	FUNCTION_BLOCK FB 347
	TITLE =G247M LOCAL COMMAND BUTTON / LAMPS GERM 8
	//COPYRIGHT:    (C) 2009  BUHLER AG, CH-9240 UZWIL, SWITZERLAND
	//
	//PRODUCT:      WinCoS_BIW01_09
	//
	//TITLE:        LOCAL COMMAND BUTTON / LAMPS GERM 8
	//                Machine group control
	//                Maschinengruppensteuerung
	//
	//--------------------------------------------------------------------------------
	//
	//IDENT:        AUTHOR:             DEPT:                              DATE:
	//
	//P01_FB347.1.0 K.Renz              CSB41                              13.Jan.2010
	//             1st Release
	//
	//--------------------------------------------------------------------------------
	//
	//PURPOSE:
	//
	//MANUAL :
	//
	//RESTRICTIONS:
	//
	//--------------------------------------------------------------------------------
	AUTHOR  : KR
	FAMILY  : USW
	VERSION : 9.9


	VAR
	  Gr       : FB10;	//Standard interface to group
	  InOutValue1    : DINT; //Data for user
	  InOutValue2    : DINT; //Data for user
	  OutWayConflict : BOOL;	//Data for user
	  OutSelectionOk : BOOL;	//Data for user
	  CmdNewValue : BOOL;	//Data for user
	  CmdNewJob   : BOOL;	//Data for user
	  OutCodeOK   : BOOL;	//Data for user
	  InEndOfJob  : BOOL ;	//Data for user
	  staWayOk      : BOOL ;	//Data for user
	  EdgeStartRelease : BOOL ;	//Data for user
	  USW8  : BOOL;	//Data for user
	  USW9 : BOOL;	//Data for user
	  USW10: BOOL;	//Data for user
	  USW11: BOOL;	//Data for user
	  USW12: BOOL;	//Data for user
	  USW13: BOOL;	//Data for user
	  USW14: BOOL;	//Data for user
	  USW15: BOOL;	//Data for user
	     #A_2811_KCL01I1 : FB14;   // DigInpCont
	     #A_2811_KCL01I2 : FB14;   // DigInpCont
	     #A_2811_KCL01I3 : FB14;   // DigInpCont
	     #A_2811_KCL01I4 : FB14;   // DigInpCont
	     #A_2811_KCL01I5 : FB14;   // DigInpCont
	     #A_2811_KCL01I6 : FB14;   // DigInpCont
	     #A_2811_KCL01O1 : FB11;   // DigOut
	     #A_2811_KCL01O2 : FB11;   // DigOut
	     #A_2815_KCL01I1 : FB14;   // DigInpCont
	     #A_2815_KCL01I2 : FB14;   // DigInpCont
	     #A_2815_KCL01I3 : FB14;   // DigInpCont
	     #A_2815_KCL01I4 : FB14;   // DigInpCont
	     #A_2815_KCL01I5 : FB14;   // DigInpCont
	     #A_2815_KCL01I6 : FB14;   // DigInpCont
	     #A_2815_KCL01I7 : FB14;   // DigInpCont
	     #A_2815_KCL01I8 : FB14;   // DigInpCont
	     #A_2815_KCL01I9 : FB14;   // DigInpCont
	     #A_2815_KCL01O1 : FB11;   // DigOut
	     #A_2815_KCL01O2 : FB11;   // DigOut
	     #A_2815_KCL01O3 : FB11;   // DigOut
	     #A_2815_KCL01O4 : FB11;   // DigOut
	     #A_2815_KCL01O5 : FB11;   // DigOut
	     #A_2815_KCL01O6 : FB11;   // DigOut
	     #A_2815_KCL01O7 : FB11;   // DigOut
	END_VAR
	VAR_TEMP
	   tmpEnable		: BOOL;
	   tmpFlag  		: BOOL;
	   tmpCmdNext		: BOOL;
	   tmpLocal  		: BOOL;
	   tmpAspOk  		: BOOL;
	   tmpHWStop 		: BOOL;
	   tmpInstanzDBNo       : INT ;
	END_VAR
	BEGIN
	NETWORK
	TITLE =
	NETWORK
	TITLE =Read command from group control
	//Parameter
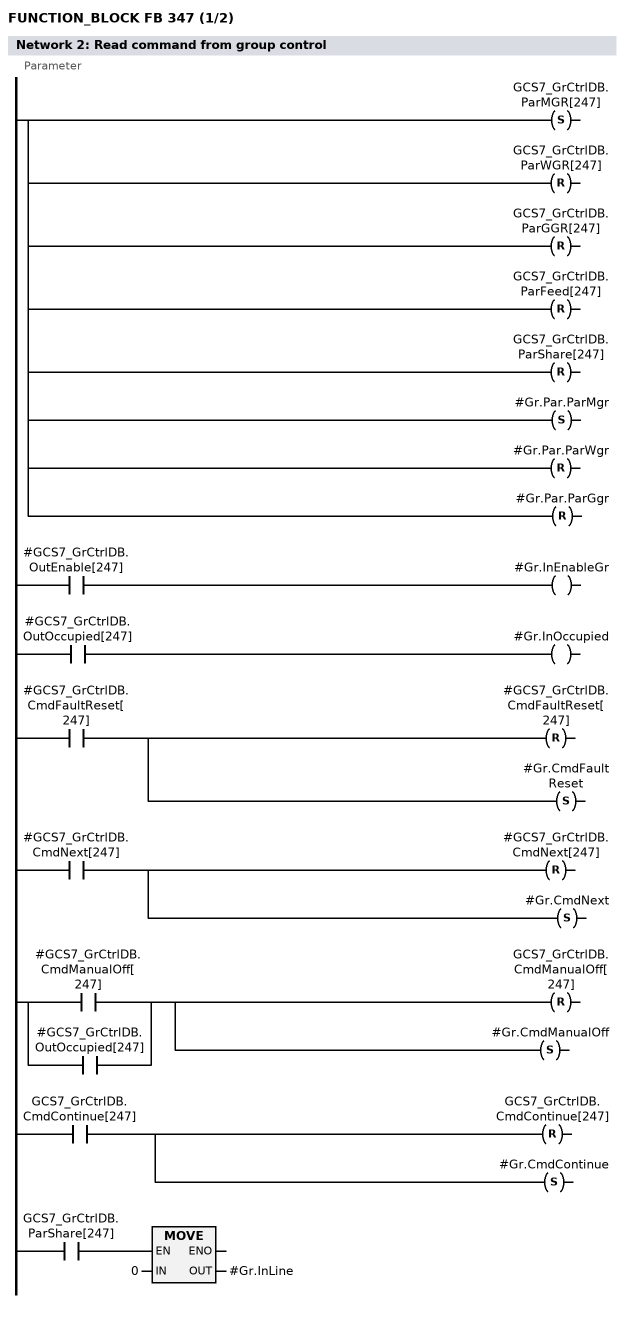
	      SET;
	      S   GCS7_GrCtrlDB.ParMGR[247];
	      R   GCS7_GrCtrlDB.ParWGR[247];
	      R   GCS7_GrCtrlDB.ParGGR[247];
	      R   GCS7_GrCtrlDB.ParFeed[247];
	      R   GCS7_GrCtrlDB.ParShare[247];
	      S   #Gr.Par.ParMgr;
	      R   #Gr.Par.ParWgr;
	      R   #Gr.Par.ParGgr;
	//Command
	      U   #GCS7_GrCtrlDB.OutEnable[247];
	      =   #Gr.InEnableGr;
	      U   #GCS7_GrCtrlDB.OutOccupied[247];
	      =   #Gr.InOccupied;
	      U   #GCS7_GrCtrlDB.CmdFaultReset[247];
	      R   #GCS7_GrCtrlDB.CmdFaultReset[247];
	      S   #Gr.CmdFaultReset;
	      U  #GCS7_GrCtrlDB.CmdNext[247];
	      R   #GCS7_GrCtrlDB.CmdNext[247];
	      S   #Gr.CmdNext;
	      U   #GCS7_GrCtrlDB.CmdManualOff[247];
	      O   #GCS7_GrCtrlDB.OutOccupied[247];
	      R   GCS7_GrCtrlDB.CmdManualOff[247];
	      S   #Gr.CmdManualOff;
	      U  GCS7_GrCtrlDB.CmdContinue[247];
	      R   GCS7_GrCtrlDB.CmdContinue[247];
	      S   #Gr.CmdContinue;
	//Init Line Number
	      U   GCS7_GrCtrlDB.ParShare[247];
	      SPBN WE00;
	      L     0;
	      T     #Gr.InLine;
	WE00: NOP   0;
	NETWORK
	TITLE =Call Methode Control
	// 1. Handle Interface PCControl
	// 2. Prepare mode --> ModePassive,ModeActive,ModeIdling
	// 3. Reset global flags of the group
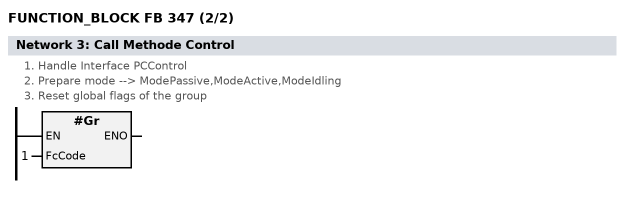
	      CALL #Gr (
	           FcCode                   := 1);
	NETWORK
	TITLE =Restart Idling Time
		L  #Gr.Par.ParIdling;
		L  2;
		>=I;
		SPB IdTm;
		T  #Gr.Par.ParIdling;
	IdTm:   NOP 0;
	      CLR;
	      S    #Gr.CmdRestartIdling;
	NETWORK
	TITLE =Prepare global flags
	NETWORK
	TITLE =Set Pattern (Target position)
	NETWORK
	TITLE =Interlocking WayOk
	//
	NETWORK
	TITLE =Interlocking Autostart
		CLR;
		R   #Gr.OutAutostart;
	NETWORK
	TITLE =Interlocking Enable
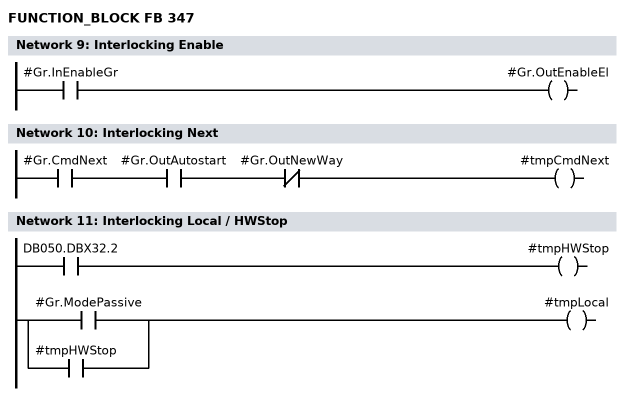
	      U     #Gr.InEnableGr;
	      =     #Gr.OutEnableEl;

	NETWORK
	TITLE =Interlocking Next
	      U     #Gr.CmdNext;
	      U     #Gr.OutAutostart;
	      UN    #Gr.OutNewWay;
	      =    #tmpCmdNext;

	NETWORK
	TITLE =Interlocking Local / HWStop
	      U    DB050.DBX32.2;
	      =    #tmpHWStop;

	      U    #Gr.ModePassive;
	      O    #tmpHWStop;
	      =    #tmpLocal;

	NETWORK
	TITLE =Interlocking Start Warning
	      NOP 0;
	//- Restart after fault --
	      U     #Gr.CmdFaultReset;
	      U     #Gr.VarFault;
	      S       "SYS_StartWarningDB".Area[9].CmdResetStartWarning;
	//- Run Timer --
	      AUF "G247M";
	      CALL  FB100 , DB100(
	       InModeHigher :=FALSE,
	       InArea     :=9,
	       InEnable   :=#Gr.OutEnableEl,
	       InLocal    :=#tmpLocal,
	       InStarted  :=#Gr.VarStarted,
	       InCmdNext  :=#tmpCmdNext,
	       OutCmdNext :=#tmpCmdNext,
	       OutStartwarning:=#Gr.VarStartWarning);
	//- Store Startwarning done  --
	//- Reset Autostart --
	      U     "SYS_StartWarningDB".TmpArea.OutStartReleaseRunningL;
	      FN    #EdgeStartRelease;
	      U     #Gr.VarFault;
	      R     #Gr.OutAutostart;
	NETWORK
	TITLE ==A-2811-KCL01I1 : SCREW ON BUTTON
	NOP 0;
	//-InLocal---
	      U     #tmpLocal;
	      =     #A_2811_KCL01I1.InLocal;
	//
	//-Monitoring---
	      CLR;
	      =      #A_2811_KCL01I1.InMonTrue;
	      CLR;
	      =      #A_2811_KCL01I1.InMonFalse;
	//
	//-PreAlarm---
	      CLR;
	      =      #A_2811_KCL01I1.InPreAlarmTrue;
	      CLR;
	      =      #A_2811_KCL01I1.InPreAlarmFalse;
	//
	//-Additional commands---
	//      CLR
	//      S     #A_2811_KCL01I1.CmdRunTimeOutTime
	//
	//-Read inputs---
	      U     E 840.4;
	      =     #A_2811_KCL01I1.InpTrue;
	      U   DB050.DBX32.2;
	      =     #A_2811_KCL01I1.InHWStop;
	       U     PLC_DPInfo.Master[1].SlavesError[84];
	       =       #A_2811_KCL01I1.InDPFault;
	//
	//-Set Parameters---
	//
	//-Call object control---
	      CALL  #A_2811_KCL01I1;
	//
	//-Write outputs---
	NETWORK
	TITLE ==A-2811-KCL01I2 : SCREW OFF BUTTON
	NOP 0;
	//-InLocal---
	      U     #tmpLocal;
	      =     #A_2811_KCL01I2.InLocal;
	//
	//-Monitoring---
	      CLR;
	      =      #A_2811_KCL01I2.InMonTrue;
	      CLR;
	      =      #A_2811_KCL01I2.InMonFalse;
	//
	//-PreAlarm---
	      CLR;
	      =      #A_2811_KCL01I2.InPreAlarmTrue;
	      CLR;
	      =      #A_2811_KCL01I2.InPreAlarmFalse;
	//
	//-Additional commands---
	//      CLR
	//      S     #A_2811_KCL01I2.CmdRunTimeOutTime
	//
	//-Read inputs---
	      U     E 840.5;
	      =     #A_2811_KCL01I2.InpTrue;
	      U   DB050.DBX32.2;
	      =     #A_2811_KCL01I2.InHWStop;
	       U     PLC_DPInfo.Master[1].SlavesError[84];
	       =       #A_2811_KCL01I2.InDPFault;
	//
	//-Set Parameters---
	//
	//-Call object control---
	      CALL  #A_2811_KCL01I2;
	//
	//-Write outputs---
	NETWORK
	TITLE ==A-2811-KCL01I3 : DRIVE FORWARD SLOWLY BUTTON
	NOP 0;
	//-InLocal---
	      U     #tmpLocal;
	      =     #A_2811_KCL01I3.InLocal;
	//
	//-Monitoring---
	      CLR;
	      =      #A_2811_KCL01I3.InMonTrue;
	      CLR;
	      =      #A_2811_KCL01I3.InMonFalse;
	//
	//-PreAlarm---
	      CLR;
	      =      #A_2811_KCL01I3.InPreAlarmTrue;
	      CLR;
	      =      #A_2811_KCL01I3.InPreAlarmFalse;
	//
	//-Additional commands---
	//      CLR
	//      S     #A_2811_KCL01I3.CmdRunTimeOutTime
	//
	//-Read inputs---
	      U     E 840.6;
	      =     #A_2811_KCL01I3.InpTrue;
	      U   DB050.DBX32.2;
	      =     #A_2811_KCL01I3.InHWStop;
	       U     PLC_DPInfo.Master[1].SlavesError[84];
	       =       #A_2811_KCL01I3.InDPFault;
	//
	//-Set Parameters---
	//
	//-Call object control---
	      CALL  #A_2811_KCL01I3;
	//
	//-Write outputs---
	NETWORK
	TITLE ==A-2811-KCL01I4 : DRIVE BACKWARD SLOWLY BUTTON
	NOP 0;
	//-InLocal---
	      U     #tmpLocal;
	      =     #A_2811_KCL01I4.InLocal;
	//
	//-Monitoring---
	      CLR;
	      =      #A_2811_KCL01I4.InMonTrue;
	      CLR;
	      =      #A_2811_KCL01I4.InMonFalse;
	//
	//-PreAlarm---
	      CLR;
	      =      #A_2811_KCL01I4.InPreAlarmTrue;
	      CLR;
	      =      #A_2811_KCL01I4.InPreAlarmFalse;
	//
	//-Additional commands---
	//      CLR
	//      S     #A_2811_KCL01I4.CmdRunTimeOutTime
	//
	//-Read inputs---
	      U     E 840.7;
	      =     #A_2811_KCL01I4.InpTrue;
	      U   DB050.DBX32.2;
	      =     #A_2811_KCL01I4.InHWStop;
	       U     PLC_DPInfo.Master[1].SlavesError[84];
	       =       #A_2811_KCL01I4.InDPFault;
	//
	//-Set Parameters---
	//
	//-Call object control---
	      CALL  #A_2811_KCL01I4;
	//
	//-Write outputs---
	NETWORK
	TITLE ==A-2811-KCL01I5 : DRIVE FORWARD FASTER BUTTON
	NOP 0;
	//-InLocal---
	      U     #tmpLocal;
	      =     #A_2811_KCL01I5.InLocal;
	//
	//-Monitoring---
	      CLR;
	      =      #A_2811_KCL01I5.InMonTrue;
	      CLR;
	      =      #A_2811_KCL01I5.InMonFalse;
	//
	//-PreAlarm---
	      CLR;
	      =      #A_2811_KCL01I5.InPreAlarmTrue;
	      CLR;
	      =      #A_2811_KCL01I5.InPreAlarmFalse;
	//
	//-Additional commands---
	//      CLR
	//      S     #A_2811_KCL01I5.CmdRunTimeOutTime
	//
	//-Read inputs---
	      U     E 841.0;
	      =     #A_2811_KCL01I5.InpTrue;
	      U   DB050.DBX32.2;
	      =     #A_2811_KCL01I5.InHWStop;
	       U     PLC_DPInfo.Master[1].SlavesError[84];
	       =       #A_2811_KCL01I5.InDPFault;
	//
	//-Set Parameters---
	//
	//-Call object control---
	      CALL  #A_2811_KCL01I5;
	//
	//-Write outputs---
	NETWORK
	TITLE ==A-2811-KCL01I6 : DRIVE BACKWARD FASTER BUTTON
	NOP 0;
	//-InLocal---
	      U     #tmpLocal;
	      =     #A_2811_KCL01I6.InLocal;
	//
	//-Monitoring---
	      CLR;
	      =      #A_2811_KCL01I6.InMonTrue;
	      CLR;
	      =      #A_2811_KCL01I6.InMonFalse;
	//
	//-PreAlarm---
	      CLR;
	      =      #A_2811_KCL01I6.InPreAlarmTrue;
	      CLR;
	      =      #A_2811_KCL01I6.InPreAlarmFalse;
	//
	//-Additional commands---
	//      CLR
	//      S     #A_2811_KCL01I6.CmdRunTimeOutTime
	//
	//-Read inputs---
	      U     E 841.1;
	      =     #A_2811_KCL01I6.InpTrue;
	      U   DB050.DBX32.2;
	      =     #A_2811_KCL01I6.InHWStop;
	       U     PLC_DPInfo.Master[1].SlavesError[84];
	       =       #A_2811_KCL01I6.InDPFault;
	//
	//-Set Parameters---
	//
	//-Call object control---
	      CALL  #A_2811_KCL01I6;
	//
	//-Write outputs---
	NETWORK
	TITLE ==A-2811-KCL01O1 : ALARM FLASHER
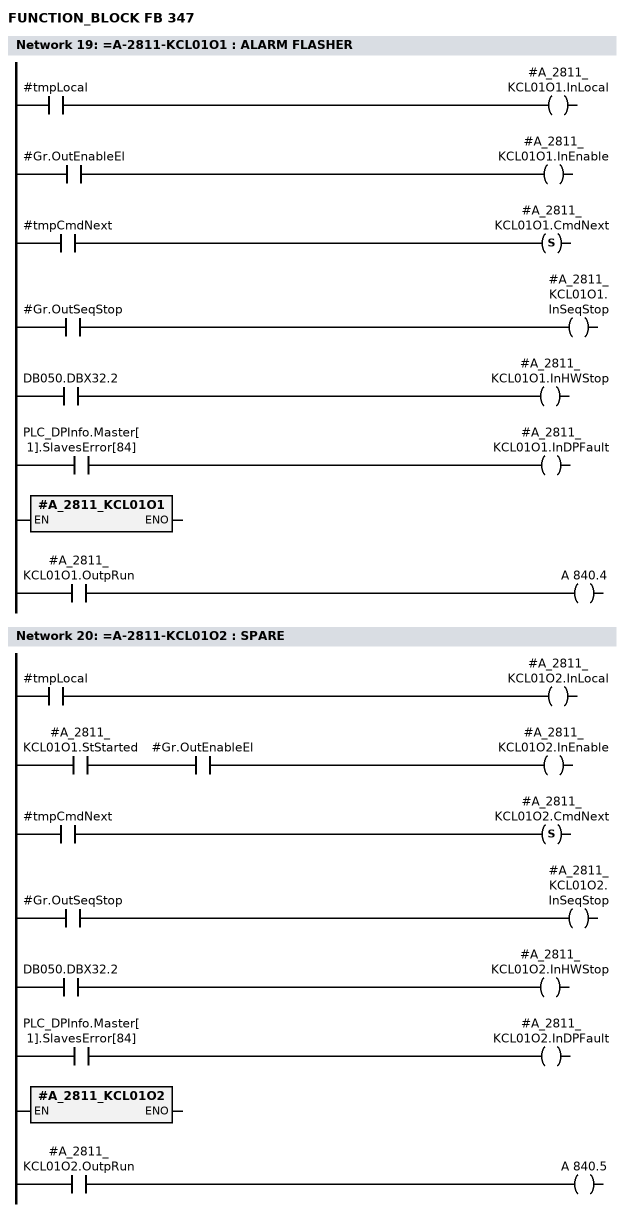
	NOP 0;
	//-InLocal---
	      U     #tmpLocal;
	      =     #A_2811_KCL01O1.InLocal;
	//
	//-Interlocking---
	      U     #Gr.OutEnableEl;
	      =     #A_2811_KCL01O1.InEnable;
	//
	      U    #tmpCmdNext;
	      S     #A_2811_KCL01O1.CmdNext;
	//
	      U     #Gr.OutSeqStop;
	      =     #A_2811_KCL01O1.InSeqStop;
	//
	//-Read inputs---
	      U   DB050.DBX32.2;
	      =     #A_2811_KCL01O1.InHWStop;
	       U     PLC_DPInfo.Master[1].SlavesError[84];
	       =       #A_2811_KCL01O1.InDPFault;
	//
	//-Set Parameters---
	//
	//-Call object control---
	      CALL  #A_2811_KCL01O1;
	//
	//-Write outputs---
	      U     #A_2811_KCL01O1.OutpRun;
	      =     A 840.4;
	NETWORK
	TITLE ==A-2811-KCL01O2 : SPARE
	NOP 0;
	//-InLocal---
	      U     #tmpLocal;
	      =     #A_2811_KCL01O2.InLocal;
	//
	//-Interlocking---
	      U     #A_2811_KCL01O1.StStarted;
	      U     #Gr.OutEnableEl;
	      =     #A_2811_KCL01O2.InEnable;
	//
	      U    #tmpCmdNext;
	      S     #A_2811_KCL01O2.CmdNext;
	//
	      U     #Gr.OutSeqStop;
	      =     #A_2811_KCL01O2.InSeqStop;
	//
	//-Read inputs---
	      U   DB050.DBX32.2;
	      =     #A_2811_KCL01O2.InHWStop;
	       U     PLC_DPInfo.Master[1].SlavesError[84];
	       =       #A_2811_KCL01O2.InDPFault;
	//
	//-Set Parameters---
	//
	//-Call object control---
	      CALL  #A_2811_KCL01O2;
	//
	//-Write outputs---
	      U     #A_2811_KCL01O2.OutpRun;
	      =     A 840.5;
	NETWORK
	TITLE ==A-2815-KCL01I1 : BACKWALL LIFTING BUTTON
	NOP 0;
	//-InLocal---
	      U     #tmpLocal;
	      =     #A_2815_KCL01I1.InLocal;
	//
	//-Monitoring---
	      CLR;
	      =      #A_2815_KCL01I1.InMonTrue;
	      CLR;
	      =      #A_2815_KCL01I1.InMonFalse;
	//
	//-PreAlarm---
	      CLR;
	      =      #A_2815_KCL01I1.InPreAlarmTrue;
	      CLR;
	      =      #A_2815_KCL01I1.InPreAlarmFalse;
	//
	//-Additional commands---
	//      CLR
	//      S     #A_2815_KCL01I1.CmdRunTimeOutTime
	//
	//-Read inputs---
	      U     E 860.0;
	      =     #A_2815_KCL01I1.InpTrue;
	      U   DB050.DBX32.2;
	      =     #A_2815_KCL01I1.InHWStop;
	       U     PLC_DPInfo.Master[1].SlavesError[85];
	       =       #A_2815_KCL01I1.InDPFault;
	//
	//-Set Parameters---
	//
	//-Call object control---
	      CALL  #A_2815_KCL01I1;
	//
	//-Write outputs---
	NETWORK
	TITLE ==A-2815-KCL01I2 : BACKWALL LOWERING BUTTON
	NOP 0;
	//-InLocal---
	      U     #tmpLocal;
	      =     #A_2815_KCL01I2.InLocal;
	//
	//-Monitoring---
	      CLR;
	      =      #A_2815_KCL01I2.InMonTrue;
	      CLR;
	      =      #A_2815_KCL01I2.InMonFalse;
	//
	//-PreAlarm---
	      CLR;
	      =      #A_2815_KCL01I2.InPreAlarmTrue;
	      CLR;
	      =      #A_2815_KCL01I2.InPreAlarmFalse;
	//
	//-Additional commands---
	//      CLR
	//      S     #A_2815_KCL01I2.CmdRunTimeOutTime
	//
	//-Read inputs---
	      U     E 860.1;
	      =     #A_2815_KCL01I2.InpTrue;
	      U   DB050.DBX32.2;
	      =     #A_2815_KCL01I2.InHWStop;
	       U     PLC_DPInfo.Master[1].SlavesError[85];
	       =       #A_2815_KCL01I2.InDPFault;
	//
	//-Set Parameters---
	//
	//-Call object control---
	      CALL  #A_2815_KCL01I2;
	//
	//-Write outputs---
	NETWORK
	TITLE ==A-2815-KCL01I3 : UNCOUPLE BUTTON
	NOP 0;
	//-InLocal---
	      U     #tmpLocal;
	      =     #A_2815_KCL01I3.InLocal;
	//
	//-Monitoring---
	      CLR;
	      =      #A_2815_KCL01I3.InMonTrue;
	      CLR;
	      =      #A_2815_KCL01I3.InMonFalse;
	//
	//-PreAlarm---
	      CLR;
	      =      #A_2815_KCL01I3.InPreAlarmTrue;
	      CLR;
	      =      #A_2815_KCL01I3.InPreAlarmFalse;
	//
	//-Additional commands---
	//      CLR
	//      S     #A_2815_KCL01I3.CmdRunTimeOutTime
	//
	//-Read inputs---
	      U     E 860.2;
	      =     #A_2815_KCL01I3.InpTrue;
	      U   DB050.DBX32.2;
	      =     #A_2815_KCL01I3.InHWStop;
	       U     PLC_DPInfo.Master[1].SlavesError[85];
	       =       #A_2815_KCL01I3.InDPFault;
	//
	//-Set Parameters---
	//
	//-Call object control---
	      CALL  #A_2815_KCL01I3;
	//
	//-Write outputs---
	NETWORK
	TITLE ==A-2815-KCL01I4 : COUPLE BUTTON
	NOP 0;
	//-InLocal---
	      U     #tmpLocal;
	      =     #A_2815_KCL01I4.InLocal;
	//
	//-Monitoring---
	      CLR;
	      =      #A_2815_KCL01I4.InMonTrue;
	      CLR;
	      =      #A_2815_KCL01I4.InMonFalse;
	//
	//-PreAlarm---
	      CLR;
	      =      #A_2815_KCL01I4.InPreAlarmTrue;
	      CLR;
	      =      #A_2815_KCL01I4.InPreAlarmFalse;
	//
	//-Additional commands---
	//      CLR
	//      S     #A_2815_KCL01I4.CmdRunTimeOutTime
	//
	//-Read inputs---
	      U     E 860.3;
	      =     #A_2815_KCL01I4.InpTrue;
	      U   DB050.DBX32.2;
	      =     #A_2815_KCL01I4.InHWStop;
	       U     PLC_DPInfo.Master[1].SlavesError[85];
	       =       #A_2815_KCL01I4.InDPFault;
	//
	//-Set Parameters---
	//
	//-Call object control---
	      CALL  #A_2815_KCL01I4;
	//
	//-Write outputs---
	NETWORK
	TITLE ==A-2815-KCL01I5 : WALL LOCKING BUTTON
	NOP 0;
	//-InLocal---
	      U     #tmpLocal;
	      =     #A_2815_KCL01I5.InLocal;
	//
	//-Monitoring---
	      CLR;
	      =      #A_2815_KCL01I5.InMonTrue;
	      CLR;
	      =      #A_2815_KCL01I5.InMonFalse;
	//
	//-PreAlarm---
	      CLR;
	      =      #A_2815_KCL01I5.InPreAlarmTrue;
	      CLR;
	      =      #A_2815_KCL01I5.InPreAlarmFalse;
	//
	//-Additional commands---
	//      CLR
	//      S     #A_2815_KCL01I5.CmdRunTimeOutTime
	//
	//-Read inputs---
	      U     E 860.4;
	      =     #A_2815_KCL01I5.InpTrue;
	      U   DB050.DBX32.2;
	      =     #A_2815_KCL01I5.InHWStop;
	       U     PLC_DPInfo.Master[1].SlavesError[85];
	       =       #A_2815_KCL01I5.InDPFault;
	//
	//-Set Parameters---
	//
	//-Call object control---
	      CALL  #A_2815_KCL01I5;
	//
	//-Write outputs---
	NETWORK
	TITLE ==A-2815-KCL01I6 : WALL UNLOCKING BUTTON
	NOP 0;
	//-InLocal---
	      U     #tmpLocal;
	      =     #A_2815_KCL01I6.InLocal;
	//
	//-Monitoring---
	      CLR;
	      =      #A_2815_KCL01I6.InMonTrue;
	      CLR;
	      =      #A_2815_KCL01I6.InMonFalse;
	//
	//-PreAlarm---
	      CLR;
	      =      #A_2815_KCL01I6.InPreAlarmTrue;
	      CLR;
	      =      #A_2815_KCL01I6.InPreAlarmFalse;
	//
	//-Additional commands---
	//      CLR
	//      S     #A_2815_KCL01I6.CmdRunTimeOutTime
	//
	//-Read inputs---
	      U     E 860.5;
	      =     #A_2815_KCL01I6.InpTrue;
	      U   DB050.DBX32.2;
	      =     #A_2815_KCL01I6.InHWStop;
	       U     PLC_DPInfo.Master[1].SlavesError[85];
	       =       #A_2815_KCL01I6.InDPFault;
	//
	//-Set Parameters---
	//
	//-Call object control---
	      CALL  #A_2815_KCL01I6;
	//
	//-Write outputs---
	NETWORK
	TITLE ==A-2815-KCL01I7 : HORIZONTAL SCREW ON BUTTON
	NOP 0;
	//-InLocal---
	      U     #tmpLocal;
	      =     #A_2815_KCL01I7.InLocal;
	//
	//-Monitoring---
	      CLR;
	      =      #A_2815_KCL01I7.InMonTrue;
	      CLR;
	      =      #A_2815_KCL01I7.InMonFalse;
	//
	//-PreAlarm---
	      CLR;
	      =      #A_2815_KCL01I7.InPreAlarmTrue;
	      CLR;
	      =      #A_2815_KCL01I7.InPreAlarmFalse;
	//
	//-Additional commands---
	//      CLR
	//      S     #A_2815_KCL01I7.CmdRunTimeOutTime
	//
	//-Read inputs---
	      U     E 860.6;
	      =     #A_2815_KCL01I7.InpTrue;
	      U   DB050.DBX32.2;
	      =     #A_2815_KCL01I7.InHWStop;
	       U     PLC_DPInfo.Master[1].SlavesError[85];
	       =       #A_2815_KCL01I7.InDPFault;
	//
	//-Set Parameters---
	//
	//-Call object control---
	      CALL  #A_2815_KCL01I7;
	//
	//-Write outputs---
	NETWORK
	TITLE ==A-2815-KCL01I8 : DIAGONAL SCREW ON BUTTON
	NOP 0;
	//-InLocal---
	      U     #tmpLocal;
	      =     #A_2815_KCL01I8.InLocal;
	//
	//-Monitoring---
	      CLR;
	      =      #A_2815_KCL01I8.InMonTrue;
	      CLR;
	      =      #A_2815_KCL01I8.InMonFalse;
	//
	//-PreAlarm---
	      CLR;
	      =      #A_2815_KCL01I8.InPreAlarmTrue;
	      CLR;
	      =      #A_2815_KCL01I8.InPreAlarmFalse;
	//
	//-Additional commands---
	//      CLR
	//      S     #A_2815_KCL01I8.CmdRunTimeOutTime
	//
	//-Read inputs---
	      U     E 860.7;
	      =     #A_2815_KCL01I8.InpTrue;
	      U   DB050.DBX32.2;
	      =     #A_2815_KCL01I8.InHWStop;
	       U     PLC_DPInfo.Master[1].SlavesError[85];
	       =       #A_2815_KCL01I8.InDPFault;
	//
	//-Set Parameters---
	//
	//-Call object control---
	      CALL  #A_2815_KCL01I8;
	//
	//-Write outputs---
	NETWORK
	TITLE ==A-2815-KCL01I9 : SCREW STOP BUTTON
	NOP 0;
	//-InLocal---
	      U     #tmpLocal;
	      =     #A_2815_KCL01I9.InLocal;
	//
	//-Monitoring---
	      CLR;
	      =      #A_2815_KCL01I9.InMonTrue;
	      CLR;
	      =      #A_2815_KCL01I9.InMonFalse;
	//
	//-PreAlarm---
	      CLR;
	      =      #A_2815_KCL01I9.InPreAlarmTrue;
	      CLR;
	      =      #A_2815_KCL01I9.InPreAlarmFalse;
	//
	//-Additional commands---
	//      CLR
	//      S     #A_2815_KCL01I9.CmdRunTimeOutTime
	//
	//-Read inputs---
	      U     E 861.0;
	      =     #A_2815_KCL01I9.InpTrue;
	      U   DB050.DBX32.2;
	      =     #A_2815_KCL01I9.InHWStop;
	       U     PLC_DPInfo.Master[1].SlavesError[85];
	       =       #A_2815_KCL01I9.InDPFault;
	//
	//-Set Parameters---
	//
	//-Call object control---
	      CALL  #A_2815_KCL01I9;
	//
	//-Write outputs---
	NETWORK
	TITLE ==A-2815-KCL01O1 : BACKWALL LIFTED
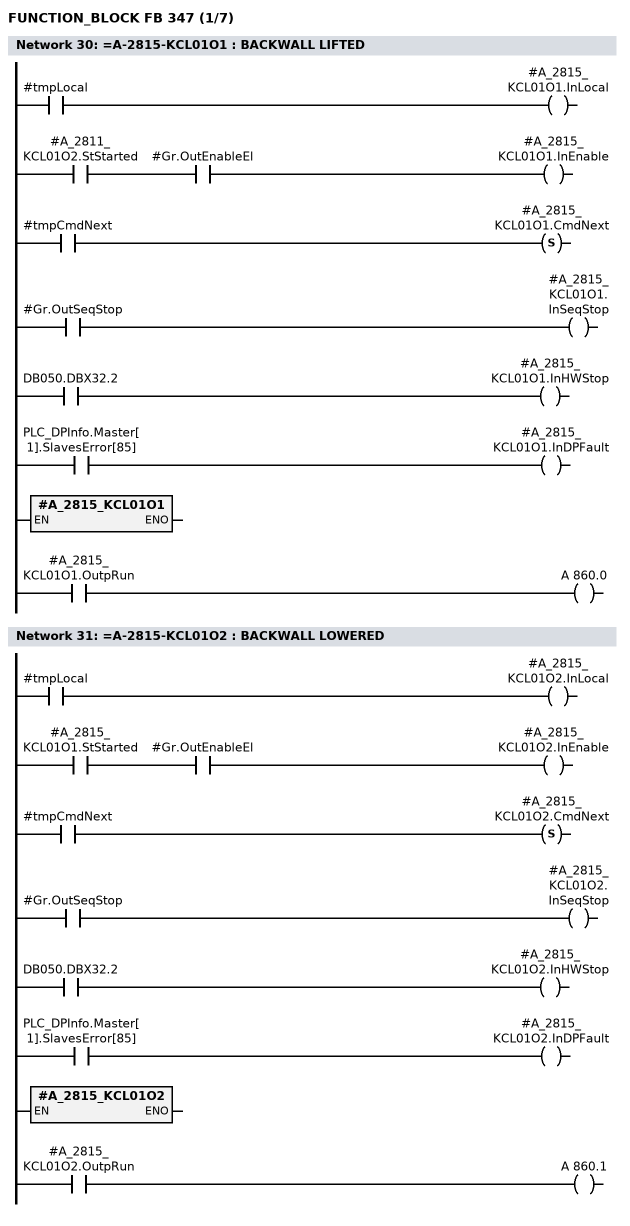
	NOP 0;
	//-InLocal---
	      U     #tmpLocal;
	      =     #A_2815_KCL01O1.InLocal;
	//
	//-Interlocking---
	      U     #A_2811_KCL01O2.StStarted;
	      U     #Gr.OutEnableEl;
	      =     #A_2815_KCL01O1.InEnable;
	//
	      U    #tmpCmdNext;
	      S     #A_2815_KCL01O1.CmdNext;
	//
	      U     #Gr.OutSeqStop;
	      =     #A_2815_KCL01O1.InSeqStop;
	//
	//-Read inputs---
	      U   DB050.DBX32.2;
	      =     #A_2815_KCL01O1.InHWStop;
	       U     PLC_DPInfo.Master[1].SlavesError[85];
	       =       #A_2815_KCL01O1.InDPFault;
	//
	//-Set Parameters---
	//
	//-Call object control---
	      CALL  #A_2815_KCL01O1;
	//
	//-Write outputs---
	      U     #A_2815_KCL01O1.OutpRun;
	      =     A 860.0;
	NETWORK
	TITLE ==A-2815-KCL01O2 : BACKWALL LOWERED
	NOP 0;
	//-InLocal---
	      U     #tmpLocal;
	      =     #A_2815_KCL01O2.InLocal;
	//
	//-Interlocking---
	      U     #A_2815_KCL01O1.StStarted;
	      U     #Gr.OutEnableEl;
	      =     #A_2815_KCL01O2.InEnable;
	//
	      U    #tmpCmdNext;
	      S     #A_2815_KCL01O2.CmdNext;
	//
	      U     #Gr.OutSeqStop;
	      =     #A_2815_KCL01O2.InSeqStop;
	//
	//-Read inputs---
	      U   DB050.DBX32.2;
	      =     #A_2815_KCL01O2.InHWStop;
	       U     PLC_DPInfo.Master[1].SlavesError[85];
	       =       #A_2815_KCL01O2.InDPFault;
	//
	//-Set Parameters---
	//
	//-Call object control---
	      CALL  #A_2815_KCL01O2;
	//
	//-Write outputs---
	      U     #A_2815_KCL01O2.OutpRun;
	      =     A 860.1;
	NETWORK
	TITLE ==A-2815-KCL01O3 : UNCOUPLED
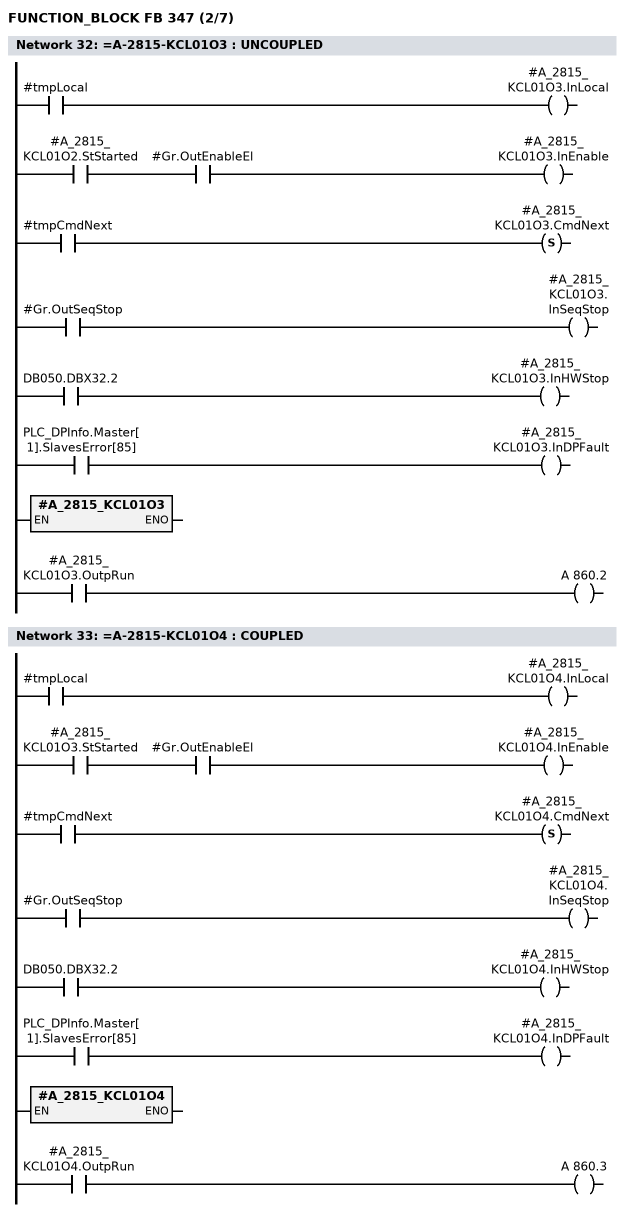
	NOP 0;
	//-InLocal---
	      U     #tmpLocal;
	      =     #A_2815_KCL01O3.InLocal;
	//
	//-Interlocking---
	      U     #A_2815_KCL01O2.StStarted;
	      U     #Gr.OutEnableEl;
	      =     #A_2815_KCL01O3.InEnable;
	//
	      U    #tmpCmdNext;
	      S     #A_2815_KCL01O3.CmdNext;
	//
	      U     #Gr.OutSeqStop;
	      =     #A_2815_KCL01O3.InSeqStop;
	//
	//-Read inputs---
	      U   DB050.DBX32.2;
	      =     #A_2815_KCL01O3.InHWStop;
	       U     PLC_DPInfo.Master[1].SlavesError[85];
	       =       #A_2815_KCL01O3.InDPFault;
	//
	//-Set Parameters---
	//
	//-Call object control---
	      CALL  #A_2815_KCL01O3;
	//
	//-Write outputs---
	      U     #A_2815_KCL01O3.OutpRun;
	      =     A 860.2;
	NETWORK
	TITLE ==A-2815-KCL01O4 : COUPLED
	NOP 0;
	//-InLocal---
	      U     #tmpLocal;
	      =     #A_2815_KCL01O4.InLocal;
	//
	//-Interlocking---
	      U     #A_2815_KCL01O3.StStarted;
	      U     #Gr.OutEnableEl;
	      =     #A_2815_KCL01O4.InEnable;
	//
	      U    #tmpCmdNext;
	      S     #A_2815_KCL01O4.CmdNext;
	//
	      U     #Gr.OutSeqStop;
	      =     #A_2815_KCL01O4.InSeqStop;
	//
	//-Read inputs---
	      U   DB050.DBX32.2;
	      =     #A_2815_KCL01O4.InHWStop;
	       U     PLC_DPInfo.Master[1].SlavesError[85];
	       =       #A_2815_KCL01O4.InDPFault;
	//
	//-Set Parameters---
	//
	//-Call object control---
	      CALL  #A_2815_KCL01O4;
	//
	//-Write outputs---
	      U     #A_2815_KCL01O4.OutpRun;
	      =     A 860.3;
	NETWORK
	TITLE ==A-2815-KCL01O5 : WALL LOCKED
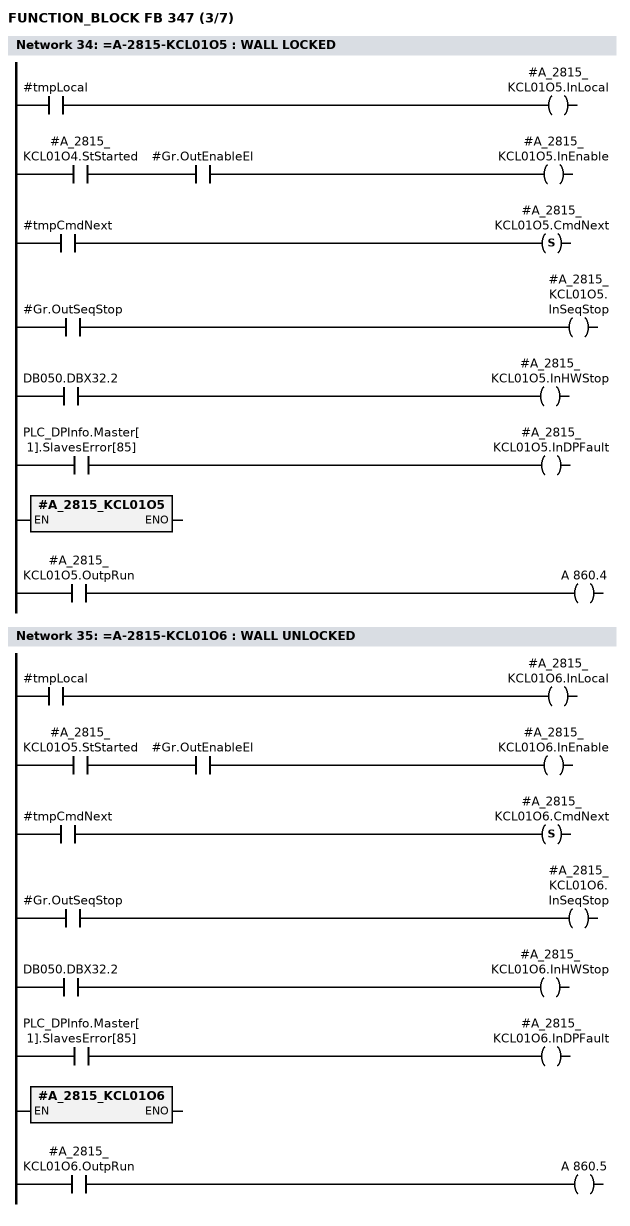
	NOP 0;
	//-InLocal---
	      U     #tmpLocal;
	      =     #A_2815_KCL01O5.InLocal;
	//
	//-Interlocking---
	      U     #A_2815_KCL01O4.StStarted;
	      U     #Gr.OutEnableEl;
	      =     #A_2815_KCL01O5.InEnable;
	//
	      U    #tmpCmdNext;
	      S     #A_2815_KCL01O5.CmdNext;
	//
	      U     #Gr.OutSeqStop;
	      =     #A_2815_KCL01O5.InSeqStop;
	//
	//-Read inputs---
	      U   DB050.DBX32.2;
	      =     #A_2815_KCL01O5.InHWStop;
	       U     PLC_DPInfo.Master[1].SlavesError[85];
	       =       #A_2815_KCL01O5.InDPFault;
	//
	//-Set Parameters---
	//
	//-Call object control---
	      CALL  #A_2815_KCL01O5;
	//
	//-Write outputs---
	      U     #A_2815_KCL01O5.OutpRun;
	      =     A 860.4;
	NETWORK
	TITLE ==A-2815-KCL01O6 : WALL UNLOCKED
	NOP 0;
	//-InLocal---
	      U     #tmpLocal;
	      =     #A_2815_KCL01O6.InLocal;
	//
	//-Interlocking---
	      U     #A_2815_KCL01O5.StStarted;
	      U     #Gr.OutEnableEl;
	      =     #A_2815_KCL01O6.InEnable;
	//
	      U    #tmpCmdNext;
	      S     #A_2815_KCL01O6.CmdNext;
	//
	      U     #Gr.OutSeqStop;
	      =     #A_2815_KCL01O6.InSeqStop;
	//
	//-Read inputs---
	      U   DB050.DBX32.2;
	      =     #A_2815_KCL01O6.InHWStop;
	       U     PLC_DPInfo.Master[1].SlavesError[85];
	       =       #A_2815_KCL01O6.InDPFault;
	//
	//-Set Parameters---
	//
	//-Call object control---
	      CALL  #A_2815_KCL01O6;
	//
	//-Write outputs---
	      U     #A_2815_KCL01O6.OutpRun;
	      =     A 860.5;
	NETWORK
	TITLE ==A-2815-KCL01O7 : CLEANING FLAP 1/2
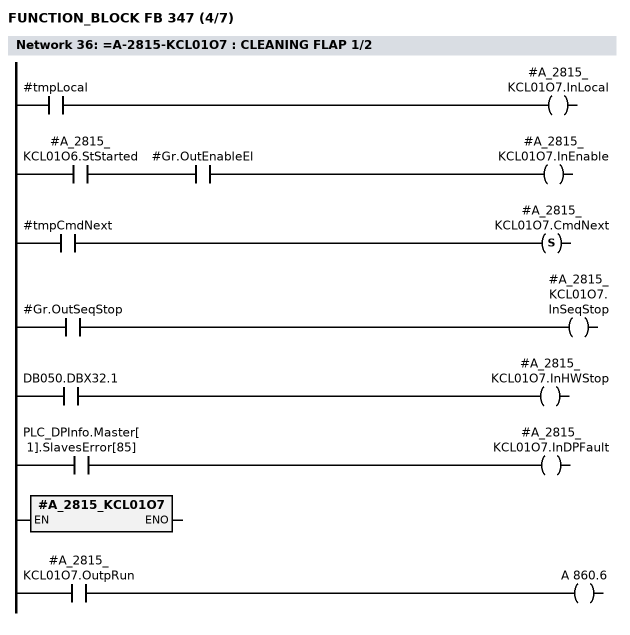
	NOP 0;
	//-InLocal---
	      U     #tmpLocal;
	      =     #A_2815_KCL01O7.InLocal;
	//
	//-Interlocking---
	      U     #A_2815_KCL01O6.StStarted;
	      U     #Gr.OutEnableEl;
	      =     #A_2815_KCL01O7.InEnable;
	//
	      U    #tmpCmdNext;
	      S     #A_2815_KCL01O7.CmdNext;
	//
	      U     #Gr.OutSeqStop;
	      =     #A_2815_KCL01O7.InSeqStop;
	//
	//-Read inputs---
	      U   DB050.DBX32.1;
	      =     #A_2815_KCL01O7.InHWStop;
	       U     PLC_DPInfo.Master[1].SlavesError[85];
	       =       #A_2815_KCL01O7.InDPFault;
	//
	//-Set Parameters---
	//
	//-Call object control---
	      CALL  #A_2815_KCL01O7;
	//
	//-Write outputs---
	      U     #A_2815_KCL01O7.OutpRun;
	      =     A 860.6;
	NETWORK
	TITLE =Test Fault
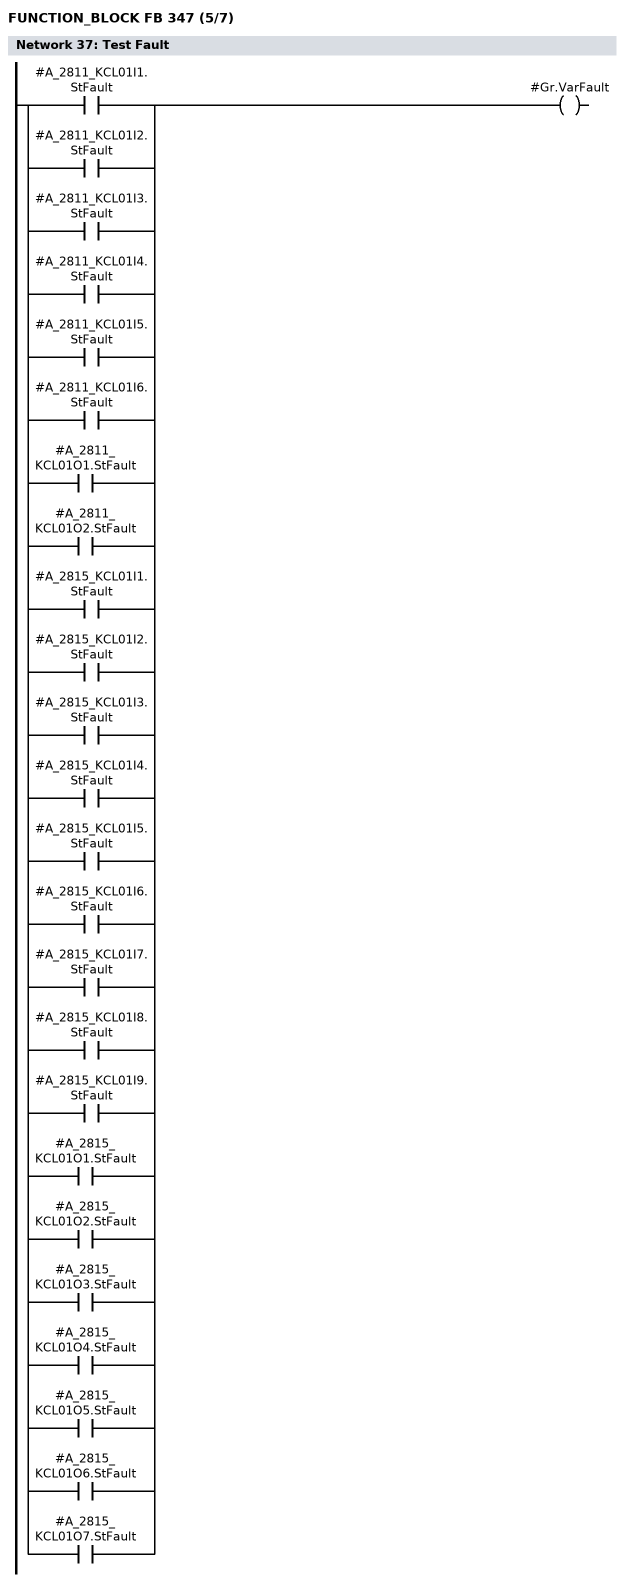
	      U     #A_2811_KCL01I1.StFault;
	      O     #A_2811_KCL01I2.StFault;
	      O     #A_2811_KCL01I3.StFault;
	      O     #A_2811_KCL01I4.StFault;
	      O     #A_2811_KCL01I5.StFault;
	      O     #A_2811_KCL01I6.StFault;
	      O     #A_2811_KCL01O1.StFault;
	      O     #A_2811_KCL01O2.StFault;
	      O     #A_2815_KCL01I1.StFault;
	      O     #A_2815_KCL01I2.StFault;
	      O     #A_2815_KCL01I3.StFault;
	      O     #A_2815_KCL01I4.StFault;
	      O     #A_2815_KCL01I5.StFault;
	      O     #A_2815_KCL01I6.StFault;
	      O     #A_2815_KCL01I7.StFault;
	      O     #A_2815_KCL01I8.StFault;
	      O     #A_2815_KCL01I9.StFault;
	      O     #A_2815_KCL01O1.StFault;
	      O     #A_2815_KCL01O2.StFault;
	      O     #A_2815_KCL01O3.StFault;
	      O     #A_2815_KCL01O4.StFault;
	      O     #A_2815_KCL01O5.StFault;
	      O     #A_2815_KCL01O6.StFault;
	      O     #A_2815_KCL01O7.StFault;
	      =     #Gr.VarFault;
	NETWORK
	TITLE =Test Warning
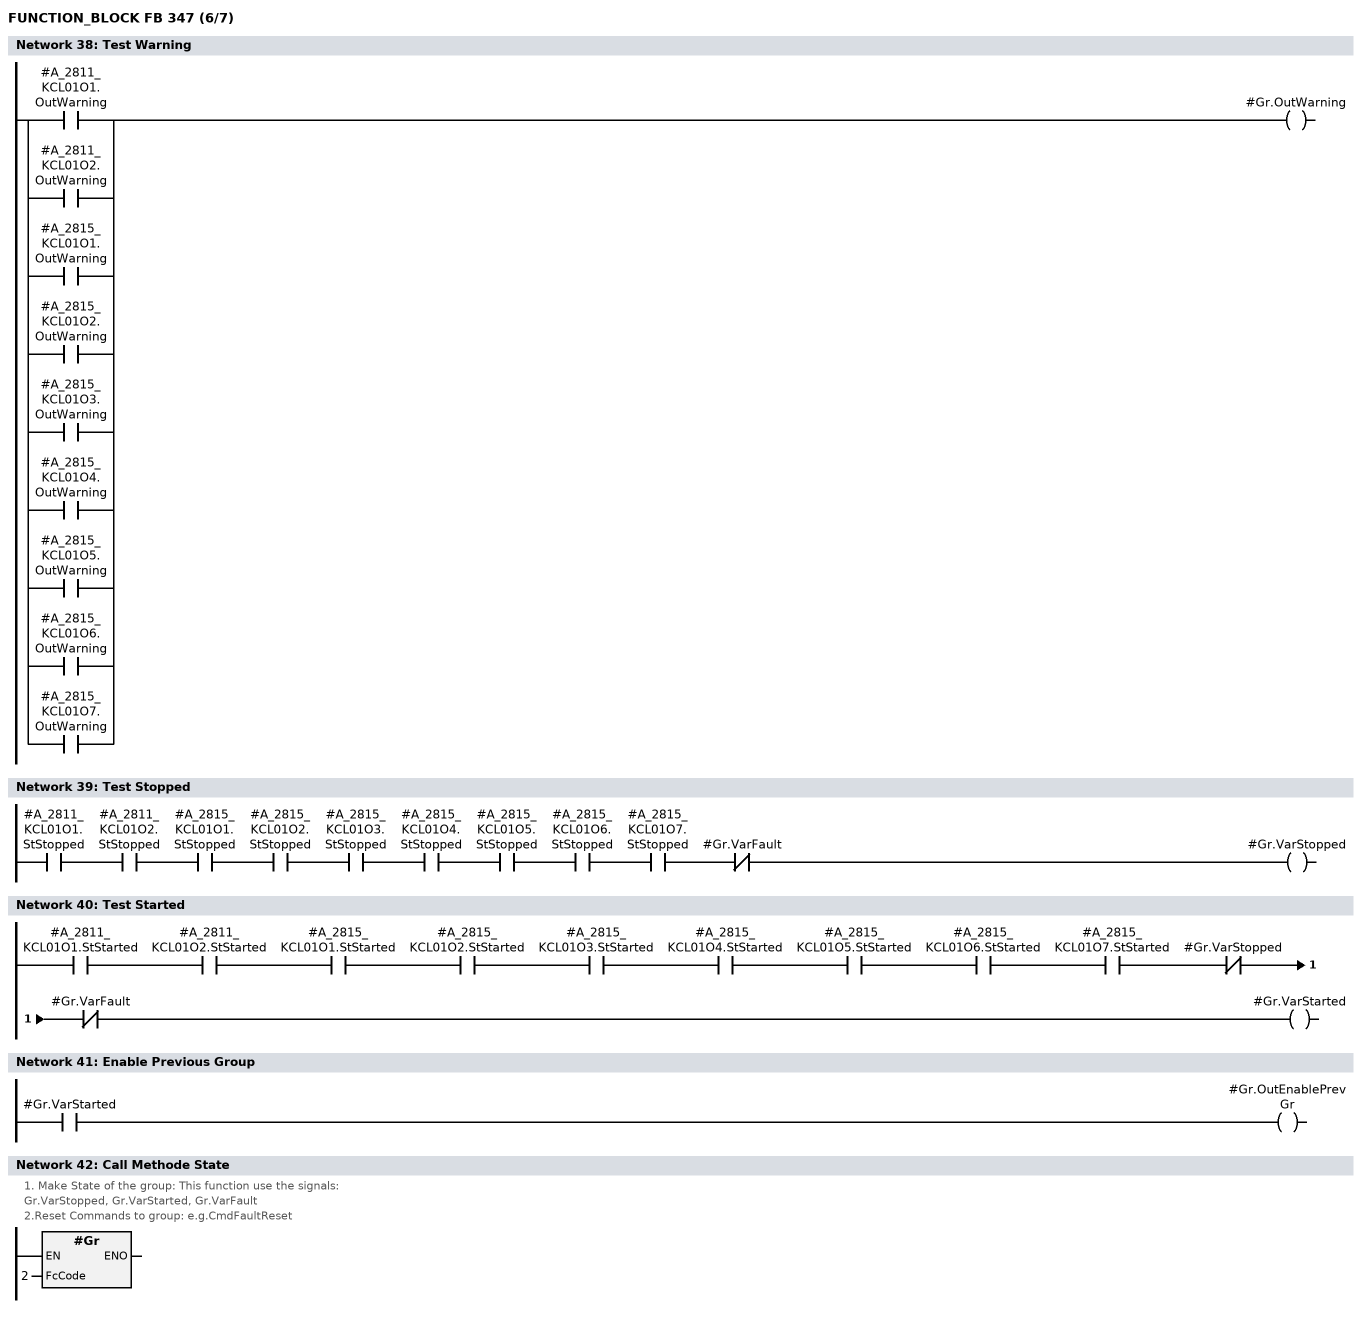
	      U     #A_2811_KCL01O1.OutWarning;
	      O     #A_2811_KCL01O2.OutWarning;
	      O     #A_2815_KCL01O1.OutWarning;
	      O     #A_2815_KCL01O2.OutWarning;
	      O     #A_2815_KCL01O3.OutWarning;
	      O     #A_2815_KCL01O4.OutWarning;
	      O     #A_2815_KCL01O5.OutWarning;
	      O     #A_2815_KCL01O6.OutWarning;
	      O     #A_2815_KCL01O7.OutWarning;
	      =     #Gr.OutWarning;
	NETWORK
	TITLE =Test Stopped
	      U     #A_2811_KCL01O1.StStopped;
	      U     #A_2811_KCL01O2.StStopped;
	      U     #A_2815_KCL01O1.StStopped;
	      U     #A_2815_KCL01O2.StStopped;
	      U     #A_2815_KCL01O3.StStopped;
	      U     #A_2815_KCL01O4.StStopped;
	      U     #A_2815_KCL01O5.StStopped;
	      U     #A_2815_KCL01O6.StStopped;
	      U     #A_2815_KCL01O7.StStopped;
	      UN   #Gr.VarFault;
	      =     #Gr.VarStopped;
	NETWORK
	TITLE =Test Started
	      U     #A_2811_KCL01O1.StStarted;
	      U     #A_2811_KCL01O2.StStarted;
	      U     #A_2815_KCL01O1.StStarted;
	      U     #A_2815_KCL01O2.StStarted;
	      U     #A_2815_KCL01O3.StStarted;
	      U     #A_2815_KCL01O4.StStarted;
	      U     #A_2815_KCL01O5.StStarted;
	      U     #A_2815_KCL01O6.StStarted;
	      U     #A_2815_KCL01O7.StStarted;
	      UN  #Gr.VarStopped;
	      UN  #Gr.VarFault;
	      =     #Gr.VarStarted;
	NETWORK
	TITLE =Enable Previous Group
	      U    #Gr.VarStarted;
	      =     #Gr.OutEnablePrevGr;
	NETWORK
	TITLE =Call Methode State
	//1. Make State of the group: This function use the signals:
	//        Gr.VarStopped, Gr.VarStarted, Gr.VarFault
	//2.Reset Commands to group: e.g.CmdFaultReset
	      CALL #Gr (
	           FcCode                   := 2);
	NETWORK
	TITLE =Init
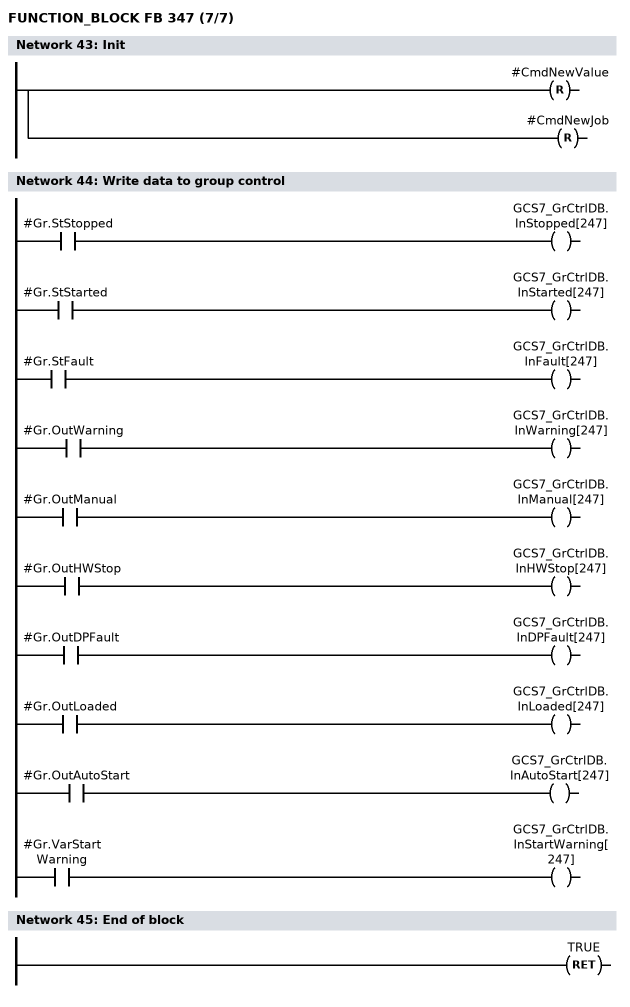
	      SET;
	      R    #CmdNewValue;
	      R    #CmdNewJob;
	NETWORK
	TITLE =Write data to group control
	      U   #Gr.StStopped;
	      =   GCS7_GrCtrlDB.InStopped[247];
	      U   #Gr.StStarted;
	      =   GCS7_GrCtrlDB.InStarted[247];
	      U   #Gr.StFault;
	      =   GCS7_GrCtrlDB.InFault[247];
	      U   #Gr.OutWarning;
	      =   GCS7_GrCtrlDB.InWarning[247];
	      U   #Gr.OutManual;
	      =   GCS7_GrCtrlDB.InManual[247];
	      U   #Gr.OutHWStop;
	      =   GCS7_GrCtrlDB.InHWStop[247];
	      U   #Gr.OutDPFault;
	      =   GCS7_GrCtrlDB.InDPFault[247];
	      U   #Gr.OutLoaded;
	      =   GCS7_GrCtrlDB.InLoaded[247];
	      U   #Gr.OutAutoStart;
	      =   GCS7_GrCtrlDB.InAutoStart[247];
	      U   #Gr.VarStartWarning;
	      =   GCS7_GrCtrlDB.InStartWarning[247];
	NETWORK
	TITLE =End of block

	BE

	END_FUNCTION_BLOCK
